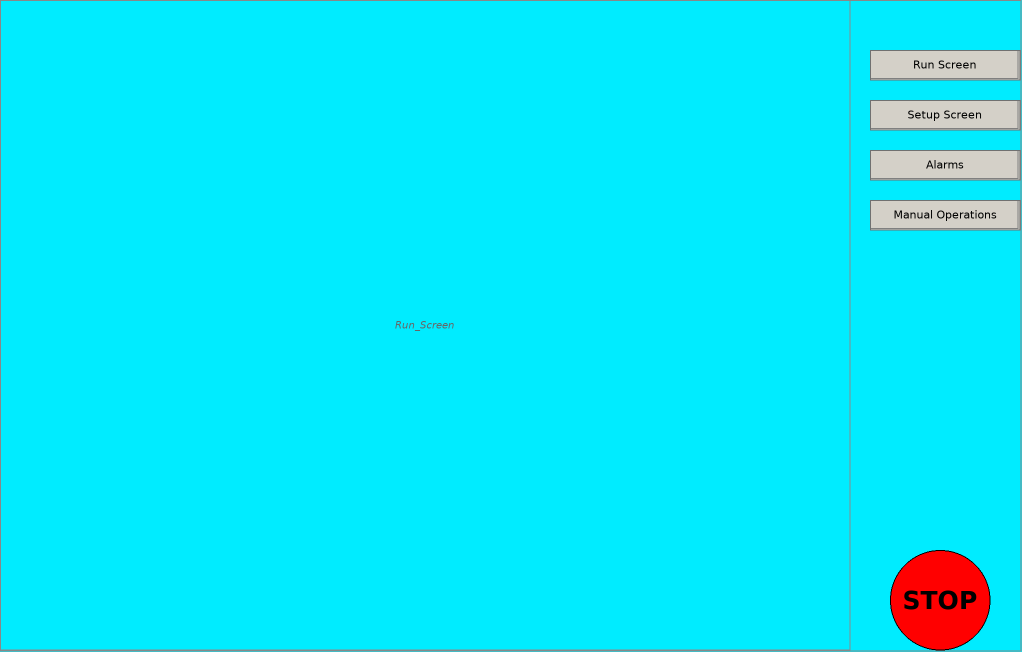
VISUALIZATION Visualization  // 1022x652
    Frame (0,0 850x650)
        shows Run_Screen()
        shows Set_Up()
        shows Alarms()
        shows Manual_Operations()
    Button (870,50 150x30), "Run Screen"
        OnMouseClick: FrameSelectionChange Selection=SelectedFrame=ea827ebc-7a9d-495a-ad7e-ffbbe3a96ee0, GlobSel=AssignType=Directly, SelType=Locally
    Button (870,100 150x30), "Setup Screen"
        OnMouseClick: FrameSelectionChange Selection=SelectedFrame=ea827ebc-7a9d-495a-ad7e-ffbbe3a96ee0, Selection=1, GlobSel=AssignType=Directly, SelType=Locally
    Button (870,150 150x30), "Alarms"
        OnMouseClick: FrameSelectionChange Selection=SelectedFrame=ea827ebc-7a9d-495a-ad7e-ffbbe3a96ee0, Selection=2, GlobSel=AssignType=Directly, SelType=Locally
    Button (870,200 150x30), "Manual Operations"
        OnMouseClick: FrameSelectionChange Selection=SelectedFrame=ea827ebc-7a9d-495a-ad7e-ffbbe3a96ee0, Selection=3, GlobSel=AssignType=Directly, SelType=Locally
    Ellipse (890,550 100x100), "RESET", invisible if: NOT :=MAIN.bStop
        OnMouseDown: toggle MAIN.bStop
    Ellipse (890,550 100x100), "STOP", invisible if: MAIN.bStop
        OnMouseDown: toggle MAIN.bStop
END_VISUALIZATION

(* stored: Version 1.1.0.1, ProductVersion 3.1.4024.0
   Visu Visualization: Id {8b4050ae-c9c7-4aba-a9be-f5ceebdef18b} *)
